PROGRAM PRG_TEST
VAR
	
fbBottleFiller_Test : FB_BottleFiller_Test;
fbBottle : FB_BottleFiller;
END_VAR


TcUnit.RUN();

END_PROGRAM

(* stored: Version 1.1.0.1, ProductVersion 3.1.4024.16
   POU PRG_TEST: Id {8d592696-06f7-48f3-8336-fe042a95e832}, SpecialFunc None *)
